Fanuc KAREL source: kt00552.KL

-- PROVISIONAL review KL for V1013-1; original PC SHA256 cab0ae9a1b5d79086a14a3ded0932cf6b34b9c1b3869b7f4f706e1e512fa01c9
-- Incomplete behavior may be omitted. Consult companion uncertainty JSON. Do not deploy.
PROGRAM KT00552
%NOLOCKGROUP
-- UNRESOLVED_DECL P1 type=000199
-- UNRESOLVED_DECL P2 type=000199
-- UNRESOLVED_DECL OUT type=000199
BEGIN
  -- UNRESOLVED_PC offsets 5-44; opcodes 49,7E,49,7E,60,7E,4A
  -- UNRESOLVED_PC offsets 49-53; opcodes 7F
END KT00552
